FUNCTION_BLOCK BasicAO (* Basic Function Block Type *)
  (* Standard: 61499-2 *)
  (* Version 0.0, 2016-04-07, 4DIAC-IDE, 4DIAC-Consortium *)
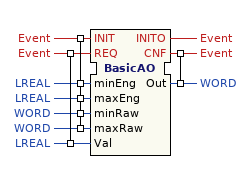
  EVENT_INPUT
    INIT WITH minEng, maxEng, minRaw, maxRaw; (* Initialization Request *)
    REQ WITH Val; (* Normal Execution Request *)
  END_EVENT
  EVENT_OUTPUT
    INITO; (* Initialization Confirm *)
    CNF WITH Out; (* Execution Confirmation *)
  END_EVENT
  VAR_INPUT
    minEng : LREAL;
    maxEng : LREAL;
    minRaw : WORD;
    maxRaw : WORD;
    Val : LREAL;
  END_VAR
  VAR_OUTPUT
    Out : WORD;
  END_VAR
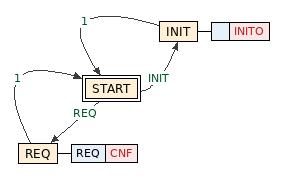
  EC_STATES
    START; (* Initial State *)
    INIT : -> INITO; (* Initialization *)
    REQ : REQ -> CNF; (* Normal execution *)
  END_STATES
  EC_TRANSITIONS
    START TO INIT := INIT;
    INIT TO START := 1;
    START TO REQ := REQ;
    REQ TO START := 1;
  END_TRANSITIONS
  ALGORITHM REQ IN ST: (* Normally executed algorithm *)
Out := LREAL_TO_WORD((Val - minEng)/(maxEng - minEng) * WORD_TO_LREAL(maxRaw - minRaw) + WORD_TO_LREAL(minRaw));
  END_ALGORITHM
END_FUNCTION_BLOCK
